FUNCTION_BLOCK TEST_Skill_varP EXTENDS FB_1_Skill
VAR_INPUT
	pUR		: POINTER TO ROBOT_UR;
	PathOfURP	: STRING := '/FNA/skill_var_point.urp';
	X: REAL := 0.5;
	Z: REAL := 0.3;
END_VAR

VAR_OUTPUT

END_VAR

VAR

    fbExecute   : R_TRIG;
    sLogMessage : STRING(255);
	phase: INT := 0;
	WaitTimer: TON;
END_VAR

// // Detect start command
// fbExecute(CLK := HMI_SKILL.bExecute);
// 
// 
// // Start / restart
// IF fbExecute.Q THEN
// 	HMI_SKILL.bExecute:=FALSE;
//     Busy := TRUE;
//     ExecutionDone:=FALSE;
// 	ExecutionResult:= NONE;
// END_IF
// 
// 
// 
// 
// // Stop immediately
// IF HMI_SKILL.bStop THEN
//     HMI_BASE.Busy:=False;
//     ExecutionDone:=TRUE;
// 	ExecutionResult:= FAILURE;
// 	phase:=0;
// 	
// 	pUR^.UR_COMM.Dashboard.Stop();
// 	HMI_SKILL.bStop:=FALSE;
// ELSE
// 
//     IF HMI_BASE.bBusy THEN
// 		IF phase=0 THEN
// 			pUR^.UR_COMM.Dashboard.LoadProgram(sPath:=PathOfURP);
// // 			pUR^.UR_COMM.Dashboard.GetLoadedProgram();
// 			phase:=1;
// 		END_IF
// 		
// 		IF phase=1 THEN
// 			IF pUR^.UR_COMM.Dashboard.LastResponseIncludes('Loading') THEN
// 				phase:=55;
// 			ELSE 
// 				pUR^.UR_COMM.Dashboard.GetLoadedProgram();
// 				phase:=44;
// 			END_IF
// 		END_IF
// 		
// 		IF phase=44 THEN
// 			IF pUR^.UR_COMM.Dashboard.LastResponseIncludes(PathOfURP) THEN
// 				phase:=55;
// 			ELSE
// 				phase:=0;
// 			END_IF
// 		END_IF
// 		
// 		//WRITE
// 		IF phase = 55 THEN
// 			pUR^.UR_COMM.RTDE.SetPoint(
// 				X  := X,
// 				Y  := 0.100,
// 				Z  := Z,
// 				Rx := 3.14,
// 				Ry := 0.0,
// 				Rz := 0.0
// 			);
// 			phase:=2;
// 		END_IF
// 		
// 		
// 		IF phase=2 THEN
// 			pUR^.UR_COMM.Dashboard.Play();
// 			phase:=3;
// 		END_IF
// 		
// 		IF phase=3 THEN
// 			IF pUR^.UR_COMM.Dashboard.LastResponseIncludes('Starting') THEN
// 				HMI_SKILL.bExecute:=FALSE;
// 				phase:=4;
// 			ELSE
// 				phase:=2;
// 			END_IF
// 		END_IF
// 		
// 		IF phase=4 THEN
// 			WaitTimer(IN:=TRUE,PT:=T#2S);
// 			IF WaitTimer.Q THEN
// 				phase:=5;
// 				WaitTimer(IN:=FALSE);
// 			END_IF
// 		END_IF
// 		
// 		IF phase=5 THEN			
// 			pUR^.UR_COMM.Dashboard.ProgramState();
// 			IF pUR^.UR_COMM.Dashboard.LastResponseIncludes('STOPPED') THEN //Skill is finished
// 				HMI_SKILL.bExecute:=FALSE;
// 				ExecutionDone:=TRUE;
// 				ExecutionResult:= SUCCESS;
// 				HMI_BASE.bBusy:=FALSE;
// 				phase:=0;
// 			END_IF
// 		END_IF
//     END_IF
// END_IF

METHOD INTERNAL StartCustomSkill : eResult

VAR
END_VAR
// !! THESE AREN'T THE METHODS YOU CALL TO START/STOP THE SKILL //
// ----- YOUR CODE HERE (incl. Alarms) -------------

HMI_SKILL.bExecute:=TRUE;


// ----- END YOUR CODE -----------------------------
ExecutionDone:=FALSE;		//IMPORTANT
ExecutionResult:=NONE;		//IMPORTANT
StartCustomSkill:=SUCCESS;
END_METHOD

METHOD INTERNAL StopCustomSkill : eResult
// !! THESE AREN'T THE METHODS YOU CALL TO START/STOP THE SKILL //
// ----- YOUR CODE HERE (incl. Alarms) -------------

HMI_SKILL.bStop:=TRUE;

// ----- END YOUR CODE -----------------------------
StopCustomSkill:=SUCCESS;
END_METHOD

END_FUNCTION_BLOCK

(* stored: Version 1.1.0.1, ProductVersion 3.1.4026.18
   POU TEST_Skill_varP: Id {cab6aeca-e3e9-45f1-83af-e9e0349cbfc5}, SpecialFunc None
   Folder Internal: Id {f208b375-b909-4557-87c5-f51552ae348b}
   Method StartCustomSkill: Id {bdb0b1c3-507b-45b3-9415-55d91fa640f0}
   Method StopCustomSkill: Id {fa598b0c-7c37-4313-9696-7420eb7696be} *)
